// TIA Portal V19 export
TYPE "PositioningMachine_Wng"
// stored: Access Published
   STRUCT
      NotAutReady { ExternalVisible := 'False'; ExternalWritable := 'False'} : Bool;
      AxisNotInOperation : Bool;
      MissingCnd_BWD { ExternalVisible := 'False'; ExternalWritable := 'False'} : Bool;
      MissingCnd_FWD { ExternalVisible := 'False'; ExternalWritable := 'False'} : Bool;
      Ax { ExternalVisible := 'False'; ExternalWritable := 'False'} : "TAx_Warnings";
   END_STRUCT;
END_TYPE
